Staubli VAL3: _plc.pgx

program _plc()
  local bool bActive
begin
  // PLC
  bActive=false
  switch plc:nToSuperV
    case 0
      //
      // Start Cycle
      //
      if taskStatus("Cycle")==-1
        cycleStatus:bToStart=true
      endIf
      bActive=true
    break
  endSwitch
  //
  if bActive
    plc:nToSuperV=-1
  endIf
end
